PROGRAM LightBulbCount
VAR
	ResetBTN: BOOL;
END_VAR

(*Counter TURN ON 5 times until LED can actually turn on*)

(*CountUp.Count (CU := LightBulb.LightSwitch, RESET := ResetBTN, PV := 5, Q=>, CV=> );

IF LightBulb.LightSwitch THEN
	LightBulb.YellowLED	:=	CountUp.Count.Q;
END_IF

*)

END_PROGRAM

(* stored: Version 1.1.0.1, ProductVersion 3.1.4024.9
   POU LightBulbCount: Id {71f65e83-10ab-48e4-a72b-032105444cab}, SpecialFunc None *)
